// TIA Portal V16 export
// export: Created 2026-03-31T12:43:22.1033848Z, ExportSetting WithDefaults, DisplayName Totally Integrated Automation Portal, DisplayVersion V16, DisplayName TIA Portal Version Control Interface, DisplayVersion V16, DisplayName TIA Portal Openness, DisplayVersion V16, DisplayName STEP 7 Professional, DisplayVersion V16, DisplayName STEP 7 Safety, DisplayVersion V16, DisplayName WinCC Advanced, DisplayVersion V16
VAR_GLOBAL   // PLC tag table "Tag table_1"
   r1 AT %M20.0 : Bool;
   tr1 AT %M20.1 : Bool;
   r2 AT %M20.2 : Bool;
   tr2 AT %M20.3 : Bool;
   r3 AT %M20.4 : Bool;
   tr3 AT %M20.5 : Bool;
   r4 AT %M20.6 : Bool;
   tr4 AT %M20.7 : Bool;
   r5 AT %M21.0 : Bool;
   tr5 AT %M21.1 : Bool;
   r6 AT %M21.2 : Bool;
   tr6 AT %M21.3 : Bool;
   r7 AT %M21.4 : Bool;
   tr7 AT %M21.5 : Bool;
   r8 AT %M21.6 : Bool;
   tr8 AT %M21.7 : Bool;
   r9 AT %M22.0 : Bool;
   tr9 AT %M22.1 : Bool;
   r10 AT %M22.2 : Bool;
   tr10 AT %M22.3 : Bool;
   r11 AT %M22.4 : Bool;
   tr11 AT %M22.5 : Bool;
   r12 AT %M22.6 : Bool;
   tr12 AT %M22.7 : Bool;
   r13 AT %M23.0 : Bool;
   tr13 AT %M23.1 : Bool;
   r14 AT %M23.2 : Bool;
   tr14 AT %M23.3 : Bool;
   r15 AT %M23.4 : Bool;
   tr15 AT %M23.5 : Bool;
END_VAR
